Fanuc KAREL source: kt00072.KL

PROGRAM KT00072
%NOLOCKGROUP
VAR
I1:INTEGER
H2 : ARRAY[2] OF SHORT
OUT:REAL
BEGIN
I1=2
H2[1]=3
OUT=((I1*H2[1]))
END KT00072
